RoboDK station: move_bill.rdk

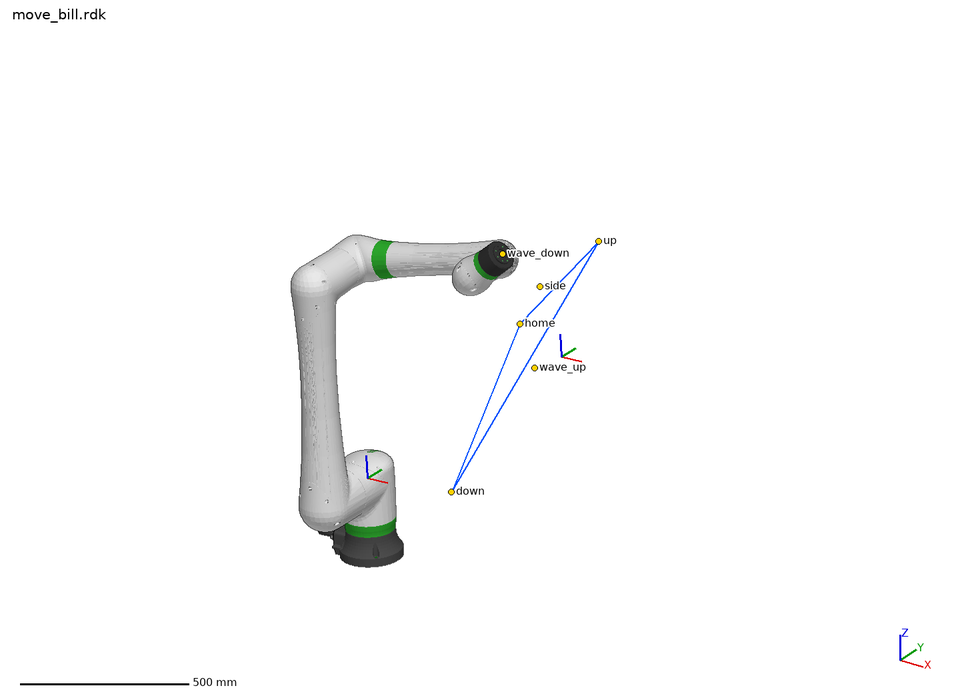
[picture v0: the station drawn from its stored meshes, robots at their saved joint values, targets as dots, program paths as lines]
Station move_bill (saved by RoboDK 5.5.4). Poses are relative to the parent item; angles as X-Y-Z fixed-axis rotations.
Station parameters (name, value as stored): LIN64
  - frame Fanuc CRX-10iA/L Base at (0, 236.15, 216.1) mm, rotated rx 0 ry -3.51 rz 0 deg
    - robot Fanuc CRX-10iA/L: 6 axes, payload 10 kg, reach 1418 mm, repeatability 0.05 mm, weight 40 kg
        modified DH rows (alpha deg, a mm, theta deg, d mm): 0, 0, 0, 245; -90, 0, -90, 0; 0, 710, 0, 0; -90, 0, 0, 540; 90, 0, 0, -150; -90, 0, 0, 160
        base shift (0, 0, -245) mm
        joint limits [-180, -180, -360, -190, -180, -190] to [180, 180, 430, 190, 180, 190]; home [0, 0, 0, 0, 0, 0]; saved at [0, 0.02, 12.35, 0, 27.239, 0]
    - frame Frame 2 at (0, 1000, 0) mm
      - target home (Cartesian target) at (700, -1150, 710) mm, rotated rx 0 ry -90 rz -180 deg; joints [0, 0, 0, 0, 0, 0] of Fanuc CRX-10iA/L
      - target down (Cartesian target) at (700, -1537.66, 317.84) mm, rotated rx 0 ry -90 rz 180 deg; joints [-36.992, 25.714, -47.037, 45.831, 57.02, -29.265] of Fanuc CRX-10iA/L
      - target up (Cartesian target) at (700, -733.87, 813.94) mm, rotated rx 0 ry -90 rz -180 deg; joints [23.782, 4.176, -4.408, 99.895, -24.163, -100.823] of Fanuc CRX-10iA/L
      - target side (Cartesian target) at (-10.61, -72.66, 254.64) mm, rotated rx 0 ry -90 rz -93.33 deg; joints [80.388, 29.718, -39.311, -170.142, -39.729, 172.388] of Fanuc CRX-10iA/L
      - target wave_up (Cartesian target) at (746, -1150, 576.73) mm, rotated rx 180 ry -70.96 rz 0 deg; joints [0, 4.887, -8.359, 0, -10.68, 0] of Fanuc CRX-10iA/L
      - target wave_down (Cartesian target) at (651.06, -1150, 927.46) mm, rotated rx 0 ry -50.41 rz -180 deg; joints [0, 0.02, 12.35, 0, 27.239, 0] of Fanuc CRX-10iA/L
  - program dance (5 instructions, listed below)
  - Python program python_move_bill (listed below)
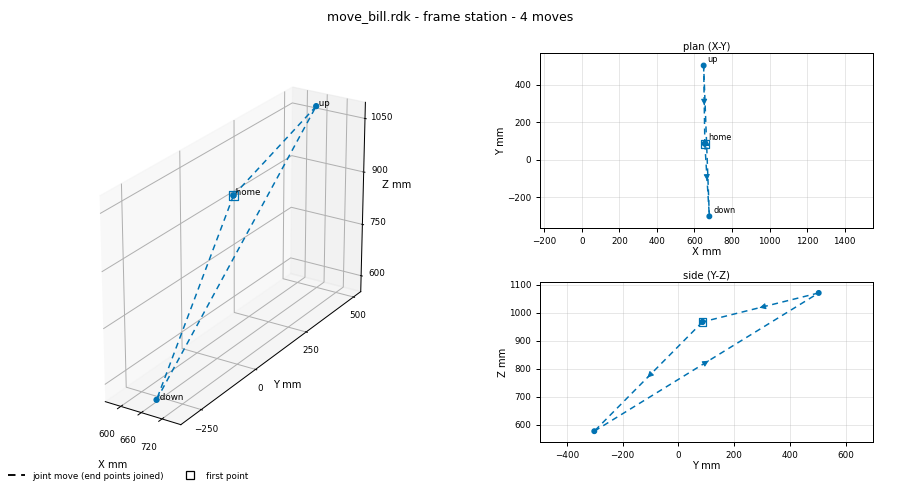
[picture p0: tool path of move_bill.rdk in frame station, 4 of 4 moves have a stored position in this frame; points joined in program order, loops and branches not executed]

--- program dance (robot Fanuc CRX-10iA/L) ---
  Set Ref.: Frame 2
  MoveJ (home)
  MoveJ (down)
  MoveJ (up)
  MoveJ (home)

--- Python program python_move_bill ---
import time

from robodk.robolink import *                  # import the robolink library
RDK = Robolink()                        # connect to the RoboDK API (RoboDK starts if it has not started

robots = RDK.ItemList(ITEM_TYPE_ROBOT)
print(robots)


# tool  = RDK.Item('SCHUNK- 1321170 Co-act EGP-C 40-N-N-KTOE_ 0')                # Get an item named Tool (name in the RoboDK station tree)

robot = RDK.Item('', ITEM_TYPE_ROBOT)   # Get the first available robot


robot.Connect()
RDK.setRunMode(RUNMODE_RUN_ROBOT)
#RDK.setRunMode(RUNMODE_SIMULATE)
#frame = RDK.ItemUserPick('Select a reference frame', ITEM_TYPE_FRAME)   # Promt the user to select a reference frame
frame = RDK.Item('Frame 2', ITEM_TYPE_FRAME)

robot.setPoseFrame(frame)
# robot.setPoseTool(tool)

# robot.setSpeed(1500)
speed = [360]

for i in range(0,len(speed)):
	print(f"Run: {i} Speed: {speed[i]}")
	RDK.ShowMessage(message = f"Run: {i} Speed: {speed[i]}")

	robot.setSpeed(speed[i], speed[i])
	robot.setSpeedJoints(speed[i])

	target = RDK.Item('home', ITEM_TYPE_TARGET)   # Get a target called "turn1"
	# target.setSpeed(speed[i])
	robot.MoveJ(target)             # Move the robot to the target using the selected reference frame

	time.sleep(1.0)

	target = RDK.Item('wave_up', ITEM_TYPE_TARGET)   # Get a target called "home"
	robot.MoveJ(target)             # Move the robot to the target using the selected reference frame

	target = RDK.Item('wave_down', ITEM_TYPE_TARGET)   # Get a target called "home"
	robot.MoveJ(target)             # Move the robot to the target using the selected reference frame



target = RDK.Item('home', ITEM_TYPE_TARGET)
robot.MoveJ(target)
